Universal Robots URScript: script_ur3e.urscript

def ur3e_dibujar():
  textmsg("=== UR3e: inicio del programa ===")

  # Guardar posición actual como HOME
  q_home = get_actual_joint_positions()
  textmsg("UR3e HOME guardado")

  # === Ir al origen calibrado del papel: UR3e ===
  textmsg("UR3e - yendo al origen calibrado")

  x0 = -0.24715
  y0 = -0.13962
  z_mesa = 0.07344
  rx = 1.36000
  ry = 2.83200
  rz = 0.00000

  movel(p[x0, y0, z_mesa+0.05000, rx, ry, rz], a=0.05, v=0.05)
  sleep(0.2)
  movel(p[x0, y0, z_mesa+0.02000, rx, ry, rz], a=0.03, v=0.003)
  sleep(0.2)
  movel(p[x0, y0, z_mesa+0.05000, rx, ry, rz], a=0.08, v=0.1)

  # === FASE 2: Dibujo - UR3e - 3 trazos ===

  # --- Trazo 1 / 3 ---
  textmsg("UR3e - Trazo 1 de 3")
  movel(p[x0+0.01457, y0+-0.00964, z_mesa+0.05000, rx, ry, rz], a=0.05, v=0.1)
  movel(p[x0+0.01457, y0+-0.00964, z_mesa+0.02000, rx, ry, rz], a=0.01, v=0.0015)
  movel(p[x0+0.01500, y0+-0.00921, z_mesa+0.02000, rx, ry, rz], a=0.008, v=0.5, r=0.0005)
  movel(p[x0+0.01714, y0+-0.00921, z_mesa+0.02000, rx, ry, rz], a=0.008, v=0.5, r=0.0005)
  movel(p[x0+0.02271, y0+-0.01136, z_mesa+0.02000, rx, ry, rz], a=0.008, v=0.5, r=0.0005)
  movel(p[x0+0.02400, y0+-0.01136, z_mesa+0.02000, rx, ry, rz], a=0.008, v=0.5, r=0.0005)
  movel(p[x0+0.02657, y0+-0.01264, z_mesa+0.02000, rx, ry, rz], a=0.008, v=0.5, r=0.0005)
  movel(p[x0+0.02871, y0+-0.01436, z_mesa+0.02000, rx, ry, rz], a=0.008, v=0.5, r=0.0005)
  movel(p[x0+0.03086, y0+-0.01693, z_mesa+0.02000, rx, ry, rz], a=0.008, v=0.5, r=0.0005)
  movel(p[x0+0.03214, y0+-0.01950, z_mesa+0.02000, rx, ry, rz], a=0.008, v=0.5, r=0.0005)
  movel(p[x0+0.03257, y0+-0.02293, z_mesa+0.02000, rx, ry, rz], a=0.008, v=0.5, r=0.0005)
  movel(p[x0+0.03300, y0+-0.02336, z_mesa+0.02000, rx, ry, rz], a=0.008, v=0.5, r=0.0005)
  movel(p[x0+0.03214, y0+-0.02850, z_mesa+0.02000, rx, ry, rz], a=0.008, v=0.5, r=0.0005)
  movel(p[x0+0.02957, y0+-0.03321, z_mesa+0.02000, rx, ry, rz], a=0.008, v=0.5, r=0.0005)
  movel(p[x0+0.02571, y0+-0.03707, z_mesa+0.02000, rx, ry, rz], a=0.008, v=0.5, r=0.0005)
  movel(p[x0+0.02314, y0+-0.03879, z_mesa+0.02000, rx, ry, rz], a=0.008, v=0.5, r=0.0005)
  movel(p[x0+0.01671, y0+-0.04093, z_mesa+0.02000, rx, ry, rz], a=0.008, v=0.5, r=0.0005)
  movel(p[x0+0.01286, y0+-0.04093, z_mesa+0.02000, rx, ry, rz], a=0.008, v=0.5, r=0.0005)
  movel(p[x0+0.00729, y0+-0.03879, z_mesa+0.02000, rx, ry, rz], a=0.008, v=0.5, r=0.0005)
  movel(p[x0+0.00343, y0+-0.03493, z_mesa+0.02000, rx, ry, rz], a=0.008, v=0.5, r=0.0005)
  movel(p[x0+0.00129, y0+-0.02979, z_mesa+0.02000, rx, ry, rz], a=0.008, v=0.5, r=0.0005)
  movel(p[x0+0.00129, y0+-0.01907, z_mesa+0.02000, rx, ry, rz], a=0.008, v=0.5, r=0.0005)
  movel(p[x0+0.00171, y0+-0.01864, z_mesa+0.02000, rx, ry, rz], a=0.008, v=0.5, r=0.0005)
  movel(p[x0+0.00600, y0+-0.01779, z_mesa+0.02000, rx, ry, rz], a=0.008, v=0.5, r=0.0005)
  movel(p[x0+0.00986, y0+-0.01564, z_mesa+0.02000, rx, ry, rz], a=0.008, v=0.5, r=0.0005)
  movel(p[x0+0.01329, y0+-0.01221, z_mesa+0.02000, rx, ry, rz], a=0.008, v=0.5, r=0.0005)
  movel(p[x0+0.01457, y0+-0.01007, z_mesa+0.02000, rx, ry, rz], a=0.008, v=0.5, r=0.0005)
  movel(p[x0+0.01457, y0+-0.01007, z_mesa+0.05000, rx, ry, rz], a=0.05, v=0.1)

  # --- Trazo 2 / 3 ---
  textmsg("UR3e - Trazo 2 de 3")
  movel(p[x0+-0.01800, y0+-0.00964, z_mesa+0.05000, rx, ry, rz], a=0.05, v=0.1)
  movel(p[x0+-0.01800, y0+-0.00964, z_mesa+0.02000, rx, ry, rz], a=0.01, v=0.0015)
  movel(p[x0+-0.01757, y0+-0.00921, z_mesa+0.02000, rx, ry, rz], a=0.008, v=0.5, r=0.0005)
  movel(p[x0+-0.01543, y0+-0.00921, z_mesa+0.02000, rx, ry, rz], a=0.008, v=0.5, r=0.0005)
  movel(p[x0+-0.01371, y0+-0.01221, z_mesa+0.02000, rx, ry, rz], a=0.008, v=0.5, r=0.0005)
  movel(p[x0+-0.01029, y0+-0.01564, z_mesa+0.02000, rx, ry, rz], a=0.008, v=0.5, r=0.0005)
  movel(p[x0+-0.00643, y0+-0.01779, z_mesa+0.02000, rx, ry, rz], a=0.008, v=0.5, r=0.0005)
  movel(p[x0+-0.00214, y0+-0.01864, z_mesa+0.02000, rx, ry, rz], a=0.008, v=0.5, r=0.0005)
  movel(p[x0+-0.00171, y0+-0.01907, z_mesa+0.02000, rx, ry, rz], a=0.008, v=0.5, r=0.0005)
  movel(p[x0+-0.00171, y0+-0.03021, z_mesa+0.02000, rx, ry, rz], a=0.008, v=0.5, r=0.0005)
  movel(p[x0+-0.00300, y0+-0.03364, z_mesa+0.02000, rx, ry, rz], a=0.008, v=0.5, r=0.0005)
  movel(p[x0+-0.00771, y0+-0.03879, z_mesa+0.02000, rx, ry, rz], a=0.008, v=0.5, r=0.0005)
  movel(p[x0+-0.01329, y0+-0.04093, z_mesa+0.02000, rx, ry, rz], a=0.008, v=0.5, r=0.0005)
  movel(p[x0+-0.01714, y0+-0.04093, z_mesa+0.02000, rx, ry, rz], a=0.008, v=0.5, r=0.0005)
  movel(p[x0+-0.01757, y0+-0.04050, z_mesa+0.02000, rx, ry, rz], a=0.008, v=0.5, r=0.0005)
  movel(p[x0+-0.02057, y0+-0.04007, z_mesa+0.02000, rx, ry, rz], a=0.008, v=0.5, r=0.0005)
  movel(p[x0+-0.02614, y0+-0.03707, z_mesa+0.02000, rx, ry, rz], a=0.008, v=0.5, r=0.0005)
  movel(p[x0+-0.03086, y0+-0.03193, z_mesa+0.02000, rx, ry, rz], a=0.008, v=0.5, r=0.0005)
  movel(p[x0+-0.03300, y0+-0.02679, z_mesa+0.02000, rx, ry, rz], a=0.008, v=0.5, r=0.0005)
  movel(p[x0+-0.03300, y0+-0.02121, z_mesa+0.02000, rx, ry, rz], a=0.008, v=0.5, r=0.0005)
  movel(p[x0+-0.03086, y0+-0.01650, z_mesa+0.02000, rx, ry, rz], a=0.008, v=0.5, r=0.0005)
  movel(p[x0+-0.02614, y0+-0.01221, z_mesa+0.02000, rx, ry, rz], a=0.008, v=0.5, r=0.0005)
  movel(p[x0+-0.01843, y0+-0.00964, z_mesa+0.02000, rx, ry, rz], a=0.008, v=0.5, r=0.0005)
  movel(p[x0+-0.01843, y0+-0.00964, z_mesa+0.05000, rx, ry, rz], a=0.05, v=0.1)

  # --- Trazo 3 / 3 ---
  textmsg("UR3e - Trazo 3 de 3")
  movel(p[x0+-0.03043, y0+0.02250, z_mesa+0.05000, rx, ry, rz], a=0.05, v=0.1)
  movel(p[x0+-0.03043, y0+0.02250, z_mesa+0.02000, rx, ry, rz], a=0.01, v=0.0015)
  movel(p[x0+-0.03000, y0+0.02293, z_mesa+0.02000, rx, ry, rz], a=0.008, v=0.5, r=0.0005)
  movel(p[x0+-0.02400, y0+0.02293, z_mesa+0.02000, rx, ry, rz], a=0.008, v=0.5, r=0.0005)
  movel(p[x0+-0.02014, y0+0.02121, z_mesa+0.02000, rx, ry, rz], a=0.008, v=0.5, r=0.0005)
  movel(p[x0+-0.01757, y0+0.01907, z_mesa+0.02000, rx, ry, rz], a=0.008, v=0.5, r=0.0005)
  movel(p[x0+-0.01157, y0+0.01093, z_mesa+0.02000, rx, ry, rz], a=0.008, v=0.5, r=0.0005)
  movel(p[x0+-0.01157, y0+0.01007, z_mesa+0.02000, rx, ry, rz], a=0.008, v=0.5, r=0.0005)
  movel(p[x0+-0.01457, y0+0.00664, z_mesa+0.02000, rx, ry, rz], a=0.008, v=0.5, r=0.0005)
  movel(p[x0+-0.01629, y0+0.00279, z_mesa+0.02000, rx, ry, rz], a=0.008, v=0.5, r=0.0005)
  movel(p[x0+-0.01629, y0+0.00107, z_mesa+0.02000, rx, ry, rz], a=0.008, v=0.5, r=0.0005)
  movel(p[x0+-0.01671, y0+0.00064, z_mesa+0.02000, rx, ry, rz], a=0.008, v=0.5, r=0.0005)
  movel(p[x0+-0.01671, y0+-0.00579, z_mesa+0.02000, rx, ry, rz], a=0.008, v=0.5, r=0.0005)
  movel(p[x0+-0.02657, y0+-0.00921, z_mesa+0.02000, rx, ry, rz], a=0.008, v=0.5, r=0.0005)
  movel(p[x0+-0.03129, y0+-0.00921, z_mesa+0.02000, rx, ry, rz], a=0.008, v=0.5, r=0.0005)
  movel(p[x0+-0.03643, y0+-0.00707, z_mesa+0.02000, rx, ry, rz], a=0.008, v=0.5, r=0.0005)
  movel(p[x0+-0.04071, y0+-0.00236, z_mesa+0.02000, rx, ry, rz], a=0.008, v=0.5, r=0.0005)
  movel(p[x0+-0.04243, y0+0.00279, z_mesa+0.02000, rx, ry, rz], a=0.008, v=0.5, r=0.0005)
  movel(p[x0+-0.04243, y0+0.00879, z_mesa+0.02000, rx, ry, rz], a=0.008, v=0.5, r=0.0005)
  movel(p[x0+-0.04157, y0+0.01179, z_mesa+0.02000, rx, ry, rz], a=0.008, v=0.5, r=0.0005)
  movel(p[x0+-0.03986, y0+0.01521, z_mesa+0.02000, rx, ry, rz], a=0.008, v=0.5, r=0.0005)
  movel(p[x0+-0.03514, y0+0.02036, z_mesa+0.02000, rx, ry, rz], a=0.008, v=0.5, r=0.0005)
  movel(p[x0+-0.03257, y0+0.02207, z_mesa+0.02000, rx, ry, rz], a=0.008, v=0.5, r=0.0005)
  movel(p[x0+-0.03086, y0+0.02250, z_mesa+0.02000, rx, ry, rz], a=0.008, v=0.5, r=0.0005)
  movel(p[x0+-0.03086, y0+0.02250, z_mesa+0.05000, rx, ry, rz], a=0.05, v=0.1)

  textmsg("UR3e - Dibujo completado")
  # === Volver a HOME ===
  textmsg("UR3e - Volviendo a HOME")
  movej(q_home, a=0.05, v=0.05)
  textmsg("UR3e - En HOME. Avisando al PC")

  # === Avisar al PC de que UR3e ha terminado ===
  socket_conn = socket_open("192.168.56.2", 50001, "pc_sync")
  if (not socket_conn):
    textmsg("UR3e - Error: No se pudo conectar con el PC en la IP: ", "192.168.56.2")
    popup("UR3e no pudo conectar con el PC. Verifica el Servidor Python.", error=True)
    halt
  else:
    socket_send_string("LISTO", "pc_sync")
    sleep(0.2)
    socket_close("pc_sync")
    textmsg("UR3e - LISTO enviado al PC correctamente")
  end

  textmsg("UR3e - Programa terminado")
end

ur3e_dibujar()
